FUNCTION BitCounter : UINT
VAR_INPUT
	fArrySize : UINT;
	fBoolArry : POINTER TO ARRAY[0..255] OF BOOL;
END_VAR
VAR
	i : UINT;			//arry pointer for thr FOR loop
	fSum_Cnt : UINT; 
END_VAR

fSum_Cnt := 0;

FOR i := 0 TO fArrySize-1 DO
	IF fBoolArry^[i] = 1
		THEN fSum_Cnt := fSum_Cnt + 1;
	END_IF
END_FOR

BitCounter := fSum_Cnt;

END_FUNCTION

(* stored: Version 1.1.0.1, ProductVersion 3.1.4024.13
   POU BitCounter: Id {7fbd3b32-a35e-4ec4-bbee-6eb33b4ebb18}, SpecialFunc None *)
